PROGRAM HeaterDuty
VAR
	
	fbTON: TON; // TON TIMER.
	
	fbTP: TP;

	pulseDuration: TIME;
END_VAR

VAR_OUTPUT
	
HeatersON:BOOL;
	
END_VAR

//This program pulses the heaters for a certain number of seconds based on the PID output

//This timer determines how often to pulse, and the max length of the pulse
//In other words, we're making a Duty Cycle
fbTON(PT := TIME#30S0MS);

//Run the pulse timer
fbTP();

//If the output of the pulse timer is true, turn on the heater valve
HeatersON:=fbTP.Q;


//Don't worry about negative values
IF TempPID.HeatingOutput >=0 THEN
	
	//Convert the output to a time (in milliseconds)
	pulseDuration:=LREAL_TO_TIME(TempPID.HeatingOutput);
	
	//Don't pulse anything shorter than 500ms.
	//It's bad for the relay
	IF pulseDuration<TIME#500MS THEN
		pulseDuration:=TIME#0MS;
	END_IF
	
	//If the durataion is greater than the max duration
	//Just turn it on and leave it on
	IF pulseDuration>fbTON.PT THEN
		HeatersON:=TRUE;
	ELSE
	
		IF fbTON.Q=TRUE THEN //when the timer is true 
			fbTP(IN:=TRUE, PT:=pulseDuration);//set the pulse length
			fbTON.IN:=FALSE;//Reset the timer funtion
		ELSE
			fbTON.IN:=TRUE; //If the timer is not true...keep timing until it is!
			fbTP.IN:=FALSE;//reset the pulse function
		END_IF
			
	END_IF

END_IF

END_PROGRAM

(* stored: Version 1.1.0.1, ProductVersion 3.1.4022.18
   POU HeaterDuty: Id {6cba3ca2-de90-475d-8ad4-7f7c5dd34981}, SpecialFunc None *)
